// TwinCAT 3 PLC project PLC1
// ProgramVersion: 3.1.4026.1+c9eadab3edd020c56c333d811d5b3c408c2550c8
// libraries:
//   Tc2_Standard, * (Beckhoff Automation GmbH)
//   Tc2_System, * (Beckhoff Automation GmbH)
// project tree:
//   / PlcTask.TcTTO
//   POUs/ FB_Alarm.TcPOU, FB_AlarmCore.TcPOU, IAlarmCore.TcIO, MAIN.TcPOU, SecondPou.TcPOU
// real-time tasks:
//   TASK PlcTask1: cycle T#10ms, priority 21, ADS port 351
//   TASK PlcTask3: cycle T#10ms, priority 23, ADS port 353

CONFIGURATION PLC1
    RESOURCE PLC ON TwinCAT3
        TASK PlcTask(INTERVAL := T#10ms, PRIORITY := 21);
        PROGRAM MAIN WITH PlcTask : MAIN;
    END_RESOURCE
END_CONFIGURATION

// ---- POUs/IAlarmCore.TcIO
INTERFACE IAlarmCore

METHOD AddAlarm
VAR_INPUT
	alarmMessage : STRING;
END_VAR
END_METHOD

//FB_Init is always available implicitly and it is used primarily for initialization.
//The return value is not evaluated. For a specific influence, you can also declare the
//methods explicitly and provide additional code there with the standard initialization
//code. You can evaluate the return value.
METHOD FB_Init: BOOL
VAR_INPUT
    bInitRetains: BOOL; // TRUE: the retain variables are initialized (reset warm / reset cold)
    bInCopyCode: BOOL;  // TRUE: the instance will be copied to the copy code afterward (online change)   
END_VAR
END_METHOD

END_INTERFACE

// ---- POUs/MAIN.TcPOU
PROGRAM MAIN
VAR
	fbAlarmCore : FB_AlarmCore;
	fbAlarm		: FB_Alarm;
	
	addAlarm	: BOOL;
END_VAR

IF addAlarm THEN
	fbAlarm.RaiseAlarm('This is Info from main program');
	addAlarm := FALSE;
END_IF

SecondUnit();

END_PROGRAM

// ---- POUs/FB_AlarmCore.TcPOU
FUNCTION_BLOCK FB_AlarmCore IMPLEMENTS IAlarmCore
VAR
	_messages				: ARRAY[1..MAXNUMBEROFALRAMS] OF STRING;
	_actualNumberOfAlarams	: UINT ;
	_alarm					: FB_Alarm;
END_VAR
VAR CONSTANT
	MAXNUMBEROFALRAMS 		: UINT := 5;
END_VAR

METHOD AddAlarm 
VAR_INPUT
	alarmMessage : STRING;
END_VAR
IF _actualNumberOfAlarams <= MAXNUMBEROFALRAMS THEN
	_messages[_actualNumberOfAlarams] := alarmMessage;
	_actualNumberOfAlarams := _actualNumberOfAlarams + 1;
END_IF
END_METHOD

//FB_Init is always available implicitly and it is used primarily for initialization.
//The return value is not evaluated. For a specific influence, you can also declare the
//methods explicitly and provide additional code there with the standard initialization
//code. You can evaluate the return value.
METHOD FB_Init: BOOL
VAR_INPUT
    bInitRetains: BOOL; // TRUE: the retain variables are initialized (reset warm / reset cold)
    bInCopyCode: BOOL;  // TRUE: the instance will be copied to the copy code afterward (online change)   
END_VAR
_actualNumberOfAlarams := 1;
_alarm.setCore(THIS^);
END_METHOD

END_FUNCTION_BLOCK

// ---- POUs/FB_Alarm.TcPOU
FUNCTION_BLOCK FB_Alarm
VAR
	_usedCore 			: IAlarmCore;
END_VAR
VAR_STAT
  	_coreSingletonInstance : IAlarmCore;
END_VAR

METHOD PRIVATE Initialize : BOOL
VAR_INPUT
END_VAR
IF (_usedCore = 0) THEN 
	_usedCore := _coreSingletonInstance; 
END_IF
END_METHOD

METHOD RaiseAlarm
VAR_INPUT
	alarmMessage : STRING;
END_VAR
Initialize();
_usedCore.AddAlarm(alarmMessage);
END_METHOD

METHOD SetCore : BOOL
VAR_INPUT
  	ref2Core : IAlarmCore; 
END_VAR
_coreSingletonInstance := ref2Core;
END_METHOD

END_FUNCTION_BLOCK

// ---- POUs/SecondPou.TcPOU
PROGRAM SecondPou
VAR
	alarm		: FB_Alarm;
	addAlarm	: BOOL;
END_VAR

IF addAlarm THEN
	alarm.RaiseAlarm('This is Info from second unit');
	addAlarm := FALSE;
END_IF

END_PROGRAM
